(* PLC project environment, Dassault Systèmes ControlBuild 2024x *)
(* stored: creationDateTime 2023-10-03T11:13:48-01:00 *)

FUNCTION_BLOCK tni_clock.environment
  VAR_INPUT
    depth : INT := 0;
  END_VAR
  VAR_IN_OUT
    B1 : BOOL := false;
    B2 : BOOL := false;
    B3 : BOOL := false;
    B4 : BOOL := false;
  END_VAR
  VAR_OUTPUT
    pressure : INT := 0;
  END_VAR
  VAR_OUTPUT
    tick : BOOL := false;
  END_VAR
  VAR
    hydrostaticPressure : REAL := 0.0;
    absolutePressure : REAL := 0.0;
  END_VAR


ACTION C_source_code:
/*********************** Pressure calculation *********************************/
/* Absolute pressure :                                                          */
/*   10 m = 2bar (1bar atm pressure and 1 bar due to water pressure)     */
/*   + 1bar every 10m                                                       */
/*                                                                             */
/* hydrostatic pressure : 1 bar every 10 m                                */
/*                                                                             */
/* 1 bar = 0.987 atm                                                           */
/*******************************************************************************/
hydrostaticPressure = (abs(depth) / 10.0) * 1024.0;
absolutePressure = hydrostaticPressure + 1024.0;

pressure = absolutePressure;



/************** Quartz management *************/
tick = ! tick;
END_ACTION
END_FUNCTION_BLOCK
